{attribute 'GeneratedUsingTerminal: EJ1914-0000-0017'}
{attribute addProperty BoxType "EJ1914-0000-0017"}
{attribute addProperty Id "Fieldvoltage_UnderrangeAT %I*BOOL1Fieldvoltage_OverrangeAT %I*BOOL1"}
{attribute addProperty CRC "2647114569"}
{attribute addProperty Size "2"}
TYPE FIELDVOLTAGE_Field_Voltage_Status_9DC7C349 :
STRUCT
	{attribute addProperty Name "Fieldvoltage_Underrange"}
	Fieldvoltage_Underrange AT %I* : BOOL;
	{attribute addProperty Name "Fieldvoltage_Overrange"}
	Fieldvoltage_Overrange AT %I* : BOOL;
END_STRUCT
END_TYPE

(* stored: Version 1.2.0.0, ProductVersion 3.1.4024.9
   DUT FIELDVOLTAGE_Field_Voltage_Status_9DC7C349: Id {2a35ae60-226d-4cf0-a73f-7e48790df379} *)
